// TIA Portal V20 export
VAR_GLOBAL   // PLC tag table "Unit1Em6"
   "BA040AZSBK20.02" AT %I1076.2 : Bool;   // STACK TABLE GAP PAD DOWN
   "BA040AZSBK20.03" AT %I1076.3 : Bool;   // STACK TABLE GAP PAD UP
   "BA040AZSBK20.06" AT %I1076.6 : Bool;   // STACK TABLE VACUUM PRESSURE SWITCH
   "BA040AZSBK20.16" AT %I1077.6 : Bool;   // STACK TABLE ELECTRODE DETECT SENSOR
   "BA030AZSSP508.02" AT %I3002.2 : Bool;   // STACK TABLE Vision STO // STO - 판정 결과때 같이 살음
   "BA030AZSSP508.03" AT %I3002.3 : Bool;   // STACK TABLE VISION JUDGMENT // TRUE = NG, FALSE= OK
   "BA040AZSPM04.00" AT %Q2012.0 : Bool;   // STACK TABLE GAP PAD UP
   "BA040AZSPM04.01" AT %Q2012.1 : Bool;   // STACK TABLE GAP PAD DOWN
   "BA040AZSPM04.02" AT %Q2012.2 : Bool;   // CATHODE MANDREL CLAMP FRONT ON
   "BA040AZSPM04.04" AT %Q2012.4 : Bool;   // CATHODE MANDREL CLAMP REAR ON
   "BA040AZSPM04.06" AT %Q2012.6 : Bool;   // ANODE MANDREL CLAMP FRONT ON
   "BA040AZSPM04.10" AT %Q2013.0 : Bool;   // ANODE MANDREL CLAMP REAR ON
   "BA040AZSBK30.04" AT %Q2104.4 : Bool;   // STACK TABLE ON
   "BA040AZSBK30.05" AT %Q2104.5 : Bool;   // STACK TABLE OFF
   "BA040AZSSP504.13" AT %Q3300.3 : Bool;   // STACK VISION CONTROLLER TRIGEER IN
END_VAR
VAR_GLOBAL CONSTANT   // user constants
   U1EM6_JOB01 : DInt := 1;
   U1EM6_JOB02 : DInt := 2;
   U1EM6_JOB03 : DInt := 3;
   U1EM6_JOB04 : DInt := 4;
   U1EM6_JOB05 : DInt := 5;
   U1EM6_JOB06 : DInt := 6;
   U1EM6_JOB07 : DInt := 7;
   U1EM6_JOB08 : DInt := 8;
   U1EM6_JOB09 : DInt := 9;
   U1EM6_JOB10 : DInt := 10;
   U1EM6_JOB11 : DInt := 11;
   U1EM6_JOB12 : DInt := 12;
   U1EM6_JOB13 : DInt := 13;
   U1EM6_JOB14 : DInt := 14;
   U1EM6_JOB15 : DInt := 15;
   U1EM6_JOB16 : DInt := 16;
   U1EM6_JOB17 : DInt := 17;
   U1EM6_JOB18 : DInt := 18;
   U1EM6_JOB19 : DInt := 19;
   U1EM6_JOB20 : DInt := 20;
   U1EM6_JOB21 : DInt := 21;
   U1EM6_JOB22 : DInt := 22;
   U1EM6_JOB23 : DInt := 23;
   U1EM6_JOB24 : DInt := 24;
   U1EM6_JOB25 : DInt := 25;
   U1EM6_JOB26 : DInt := 26;
   U1EM6_JOB27 : DInt := 27;
   U1EM6_JOB28 : DInt := 28;
   U1EM6_JOB29 : DInt := 29;
   U1EM6_JOB30 : DInt := 30;
   U1EM6_JOB31 : DInt := 31;
   U1EM6_JOB32 : DInt := 32;
   U1EM6_JOB33 : DInt := 33;
   U1EM6_JOB34 : DInt := 34;
   U1EM6_JOB35 : DInt := 35;
   U1EM6_JOB36 : DInt := 36;
   U1EM6_JOB37 : DInt := 37;
   U1EM6_JOB38 : DInt := 38;
   U1EM6_JOB39 : DInt := 39;
   U1EM6_JOB40 : DInt := 40;
   U1EM6_JOB41 : DInt := 41;
   U1EM6_JOB42 : DInt := 42;
   U1EM6_JOB43 : DInt := 43;
   U1EM6_JOB44 : DInt := 44;
   U1EM6_JOB45 : DInt := 45;
   U1EM6_JOB46 : DInt := 46;
   U1EM6_JOB47 : DInt := 47;
   U1EM6_JOB48 : DInt := 48;
   U1EM6_JOB49 : DInt := 49;
   U1EM6_JOB50 : DInt := 50;
   U1EM6_JOB51 : DInt := 51;
   U1EM6_JOB52 : DInt := 52;
   U1EM6_JOB53 : DInt := 53;
   U1EM6_JOB54 : DInt := 54;
   U1EM6_JOB55 : DInt := 55;
   U1EM6_JOB56 : DInt := 56;
   U1EM6_JOB57 : DInt := 57;
   U1EM6_JOB58 : DInt := 58;
   U1EM6_JOB59 : DInt := 59;
   U1EM6_JOB60 : DInt := 60;
   U1EM6_JOB61 : DInt := 61;
   U1EM6_JOB62 : DInt := 62;
   U1EM6_JOB63 : DInt := 63;
   U1EM6_JOB64 : DInt := 64;
   U1EM6_JOB65 : DInt := 65;
   U1EM6_JOB66 : DInt := 66;
   U1EM6_JOB67 : DInt := 67;
   U1EM6_JOB68 : DInt := 68;
   U1EM6_JOB69 : DInt := 69;
   U1EM6_JOB70 : DInt := 70;
   U1EM6_JOB71 : DInt := 71;
   U1EM6_JOB72 : DInt := 72;
   U1EM6_JOB73 : DInt := 73;
   U1EM6_JOB74 : DInt := 74;
   U1EM6_JOB75 : DInt := 75;
   U1EM6_JOB76 : DInt := 76;
   U1EM6_JOB77 : DInt := 77;
   U1EM6_JOB78 : DInt := 78;
   U1EM6_JOB79 : DInt := 79;
   U1EM6_JOB80 : DInt := 80;
   U1EM6_JOB81 : DInt := 81;
   U1EM6_JOB82 : DInt := 82;
   U1EM6_JOB83 : DInt := 83;
   U1EM6_JOB84 : DInt := 84;
   U1EM6_JOB85 : DInt := 85;
   U1EM6_JOB86 : DInt := 86;
   U1EM6_JOB87 : DInt := 87;
   U1EM6_JOB88 : DInt := 88;
   U1EM6_JOB89 : DInt := 89;
   U1EM6_JOB90 : DInt := 90;
   U1EM6_JOB91 : DInt := 91;
   U1EM6_JOB92 : DInt := 92;
   U1EM6_JOB93 : DInt := 93;
   U1EM6_JOB94 : DInt := 94;
   U1EM6_JOB95 : DInt := 95;
   U1EM6_JOB96 : DInt := 96;
   U1EM6_JOB97 : DInt := 97;
   U1EM6_JOB98 : DInt := 98;
   U1EM6_JOB99 : DInt := 99;
   U1EM6_SEQUENCE01 : Int := 1;
   U1EM6_SEQUENCE02 : Int := 2;
   U1EM6_SEQUENCE03 : Int := 3;
   U1EM6_SEQUENCE04 : Int := 4;
   U1EM6_SEQUENCE05 : Int := 5;
   U1EM6_SEQUENCE06 : Int := 6;
   U1EM6_SEQUENCE07 : Int := 7;
   U1EM6_SEQUENCE08 : Int := 8;
   U1EM6_SEQUENCE09 : Int := 9;
   U1EM6_SEQUENCE10 : Int := 10;
   U1EM6_SEQUENCE11 : Int := 11;
   U1EM6_SEQUENCE12 : Int := 12;
   U1EM6_SEQUENCE13 : Int := 13;
   U1EM6_SEQUENCE14 : Int := 14;
   U1EM6_SEQUENCE15 : Int := 15;
   U1EM6_SEQUENCE16 : Int := 16;
   U1EM6_SEQUENCE17 : Int := 17;
   U1EM6_SEQUENCE18 : Int := 18;
   U1EM6_SEQUENCE19 : Int := 19;
   U1EM6_SEQUENCE20 : Int := 20;
   U1EM6_SEQUENCE21 : Int := 21;
   U1EM6_SEQUENCE22 : Int := 22;
   U1EM6_SEQUENCE23 : Int := 23;
   U1EM6_SEQUENCE24 : Int := 24;
   U1EM6_SEQUENCE25 : Int := 25;
   U1EM6_SEQUENCE26 : Int := 26;
   U1EM6_SEQUENCE27 : Int := 27;
   U1EM6_SEQUENCE28 : Int := 28;
   U1EM6_SEQUENCE29 : Int := 29;
   U1EM6_SEQUENCE30 : Int := 30;
   U1EM6_SEQUENCE31 : Int := 31;
   U1EM6_SEQUENCE32 : Int := 32;
   U1EM6_SEQUENCE33 : Int := 33;
   U1EM6_SEQUENCE34 : Int := 34;
   U1EM6_SEQUENCE35 : Int := 35;
   U1EM6_SEQUENCE36 : Int := 36;
   U1EM6_SEQUENCE37 : Int := 37;
   U1EM6_SEQUENCE38 : Int := 38;
   U1EM6_SEQUENCE39 : Int := 39;
   U1EM6_SEQUENCE40 : Int := 40;
   U1EM6_SEQUENCE41 : Int := 41;
   U1EM6_SEQUENCE42 : Int := 42;
   U1EM6_SEQUENCE43 : Int := 43;
   U1EM6_SEQUENCE44 : Int := 44;
   U1EM6_SEQUENCE45 : Int := 45;
   U1EM6_SEQUENCE46 : Int := 46;
   U1EM6_SEQUENCE47 : Int := 47;
   U1EM6_SEQUENCE48 : Int := 48;
   U1EM6_SEQUENCE49 : Int := 49;
   U1EM6_SEQUENCE50 : Int := 50;
   U1EM6_SEQUENCE51 : Int := 51;
   U1EM6_SEQUENCE52 : Int := 52;
   U1EM6_SEQUENCE53 : Int := 53;
   U1EM6_SEQUENCE54 : Int := 54;
   U1EM6_SEQUENCE55 : Int := 55;
   U1EM6_SEQUENCE56 : Int := 56;
   U1EM6_SEQUENCE57 : Int := 57;
   U1EM6_SEQUENCE58 : Int := 58;
   U1EM6_SEQUENCE59 : Int := 59;
   U1EM6_SEQUENCE60 : Int := 60;
   U1EM6_SEQUENCE61 : Int := 61;
   U1EM6_SEQUENCE62 : Int := 62;
   U1EM6_SEQUENCE63 : Int := 63;
   U1EM6_SEQUENCE64 : Int := 64;
   U1EM6_SEQUENCE65 : Int := 65;
   U1EM6_SEQUENCE66 : Int := 66;
   U1EM6_SEQUENCE67 : Int := 67;
   U1EM6_SEQUENCE68 : Int := 68;
   U1EM6_SEQUENCE69 : Int := 69;
   U1EM6_SEQUENCE70 : Int := 70;
   U1EM6_SEQUENCE71 : Int := 71;
   U1EM6_SEQUENCE72 : Int := 72;
   U1EM6_SEQUENCE73 : Int := 73;
   U1EM6_SEQUENCE74 : Int := 74;
   U1EM6_SEQUENCE75 : Int := 75;
   U1EM6_SEQUENCE76 : Int := 76;
   U1EM6_SEQUENCE77 : Int := 77;
   U1EM6_SEQUENCE78 : Int := 78;
   U1EM6_SEQUENCE79 : Int := 79;
   U1EM6_SEQUENCE80 : Int := 80;
   U1EM6_SEQUENCE81 : Int := 81;
   U1EM6_SEQUENCE82 : Int := 82;
   U1EM6_SEQUENCE83 : Int := 83;
   U1EM6_SEQUENCE84 : Int := 84;
   U1EM6_SEQUENCE85 : Int := 85;
   U1EM6_SEQUENCE86 : Int := 86;
   U1EM6_SEQUENCE87 : Int := 87;
   U1EM6_SEQUENCE88 : Int := 88;
   U1EM6_SEQUENCE89 : Int := 89;
   U1EM6_SEQUENCE90 : Int := 90;
   U1EM6_SEQUENCE91 : Int := 91;
   U1EM6_SEQUENCE92 : Int := 92;
   U1EM6_SEQUENCE93 : Int := 93;
   U1EM6_SEQUENCE94 : Int := 94;
   U1EM6_SEQUENCE95 : Int := 95;
   U1EM6_SEQUENCE96 : Int := 96;
   U1EM6_SEQUENCE97 : Int := 97;
   U1EM6_SEQUENCE98 : Int := 98;
   U1EM6_SEQUENCE99 : Int := 99;
   U1EM6_NO_OF_SEQUENCE : USInt := 3;
   U1EM6_NO_OF_AXES : USInt := 14;
   U1EM6_NO_OF_CAMS : USInt := 18;
   U1EM6_NO_OF_OUTPUTCAM : USInt := 6;
END_VAR
